{attribute 'qualified_only'}
{attribute 'strict'}
TYPE eServiceModuleSTM :
(
	Waiting,
	Running,
	PostRunning,
	PreparingForError
);
END_TYPE

(* stored: Version 1.1.0.1, ProductVersion 3.1.4024.12
   DUT eServiceModuleSTM: Id {2a699666-39b1-4315-8ecf-19f90afb5acd} *)
